TYPE TcoKrc4_Outputs_v_5_x_x :
STRUCT
    Outputs AT %Q* : ARRAY[0..63] OF BYTE;
END_STRUCT
END_TYPE

(* stored: Version 1.1.0.1, ProductVersion 3.1.4024.12
   DUT TcoKrc4_Outputs_v_5_x_x: Id {be1b8d63-aacf-02f9-003a-363dcfc5d318} *)
